Staubli VAL3: config.dtx

public bool bLog
public mdesc mNomSpeed = {blend=off}
public num nLOGDETECT = 1
public num nLOGMISC = 8
public num nLOGMOTION = 2
public num nLOGQUEUE = 4
public num nLog = 2
public num nMAXCONVEYOR = 30
public string sGENERICCONV = "GenericConv"
public string sGEOMETRYLIB = "Geometry"
public string sGEOMETRYLIB_RS = "GeometryRS"
string sPATH
public string sPATHCONVEYOR = "Disk://Tracking\Conveyors\"
public string sPATHDETECTION = "Disk://Tracking\Detections\"
public string sPATHENCODER = "Disk://Tracking\Encoders\"
public string sPATHLANGUAGE = "Disk://Tracking\language\"
public string sPATHTEMPLATE = "Disk://Tracking\Templates\"
public string sSETTINGPATH = "Disk://Tracking\language\english\"
public string sVERSION = "s7.4.0"
public tool tPointer = {z=130, fatherId=flange[0], ioLink=valve1}
public trsf trApproach = {z=-30}
